{attribute 'GeneratedUsingTerminal: EK1100-0000-0018'}
{attribute addProperty BoxType "EK1100-0000-0018"}
{attribute addProperty Id "RC70_B1_EL7041_1000EL7041_86DE63E743RC70_B2_EL7041_1000EL7041_86DE63E743RC70_C11_EL7041_1000EL7041_86DE63E743RC70_C12_EL7041_1000EL7041_86DE63E743RC70_C21_EL7041_1000EL7041_86DE63E743RC70_C22_EL7041_1000EL7041_86DE63E743RC70_2_EndTerminal_EL9010EL9010_D29C20850"}
{attribute addProperty CRC "3588068977"}
{attribute addProperty Size "258"}
{attribute addProperty Name "RC70_2 (EK1100)"}
TYPE RC70_2_EK1100_D5DD9671 EXTENDS EK1100_1FC0878B :
STRUCT
	{attribute addProperty Name "RC70_B1 (EL7041-1000)"}
	{attribute addProperty PreviousPort "RC70_2 (EK1100) : B"}
	RC70_B1_EL7041_1000 : EL7041_86DE63E7;
	{attribute addProperty Name "RC70_B2 (EL7041-1000)"}
	{attribute addProperty PreviousPort "RC70_B1 (EL7041-1000) : B"}
	RC70_B2_EL7041_1000 : EL7041_86DE63E7;
	{attribute addProperty Name "RC70_C11 (EL7041-1000)"}
	{attribute addProperty PreviousPort "RC70_B2 (EL7041-1000) : B"}
	RC70_C11_EL7041_1000 : EL7041_86DE63E7;
	{attribute addProperty Name "RC70_C12 (EL7041-1000)"}
	{attribute addProperty PreviousPort "RC70_C11 (EL7041-1000) : B"}
	RC70_C12_EL7041_1000 : EL7041_86DE63E7;
	{attribute addProperty Name "RC70_C21 (EL7041-1000)"}
	{attribute addProperty PreviousPort "RC70_C12 (EL7041-1000) : B"}
	RC70_C21_EL7041_1000 : EL7041_86DE63E7;
	{attribute addProperty Name "RC70_C22 (EL7041-1000)"}
	{attribute addProperty PreviousPort "RC70_C21 (EL7041-1000) : B"}
	RC70_C22_EL7041_1000 : EL7041_86DE63E7;
	{attribute addProperty Name "RC70_2_EndTerminal (EL9010)"}
	{attribute addProperty PreviousPort "RC70_C22 (EL7041-1000) : B"}
	RC70_2_EndTerminal_EL9010 : EL9010_D29C2085;
END_STRUCT
END_TYPE

(* stored: Version 1.2.0.0, ProductVersion 3.1.4024.11
   DUT RC70_2_EK1100_D5DD9671: Id {3327fe38-f015-0e20-03d8-a8701d947ef7} *)
